% RSLogix 500 project FAIL SAFE_BAK000.RSS, saved by version 10.00.00.00 %
PROJECT "UNTITLED"    % processor: Bul.1763 MicroLogix 1100 Series B %

PROGRAM FILES
  LAD 2 "FAIL SAFE"  3 rungs
  LAD 3 "MAIN"  2 rungs

DATA FILES
  O0 OUTPUT  4 elements
  I1 INPUT  6 elements
  S2 STATUS  66 elements
  B3 BINARY  1 elements
  T4 TIMER  1 elements
  C5 COUNTER  1 elements
  R6 CONTROL  1 elements
  N7 INTEGER  1 elements
  F8 FLOAT  1 elements

LADDER 2 "FAIL SAFE"
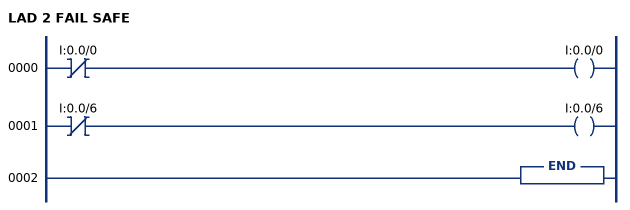
% Rung: 0 %
SOR XIO I:0.0/0 OTE I:0.0/0 EOR
% Rung: 1 %
SOR XIO I:0.0/6 OTE I:0.0/6 EOR
% Rung: 2 %
SOR END EOR

LADDER 3 "MAIN"
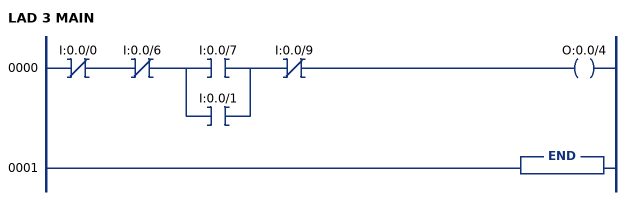
% Rung: 0 %
SOR XIO I:0.0/0 XIO I:0.0/6 BST XIC I:0.0/7 NXB XIC I:0.0/1 BND XIO I:0.0/9 OTE O:0.0/4 EOR
% Rung: 1 %
SOR END EOR
